DATA_BLOCK "PID_Feeder_4"
{InstructionName := 'PID_Compact';
 LibVersion := '1.2';
 S7_Optimized_Access := 'TRUE' }
AUTHOR : SIMATIC
NAME : PID_Cmpt
VERSION : 1.2
NON_RETAIN
PID_Compact

BEGIN
   sby_EsData_1 := 16#01;
   si_Unit := 1;
   si_Type := 9;
   sPid_Cmpt.b_Input_PER_On := FALSE;
   sPid_Cmpt.r_Pv_Hlm := 10000.0;
   sPid_Cmpt.r_Pv_Llm := -20.0;
   sPid_Cmpt.r_Pv_HWrn := 10000.0;
   sPid_Cmpt.r_Pv_LWrn := 0.0;
   sRet.r_Ctrl_Gain := 0.007823471;
   sRet.r_Ctrl_Ti := 0.3854144;
   sRet.r_Ctrl_Td := 0.04731367;
   sRet.r_Ctrl_A := 0.1;
   sRet.r_Ctrl_B := 1.0;
   sRet.r_Ctrl_Cycle := 0.1000067;

END_DATA_BLOCK

